FUNCTION_BLOCK C_BINARYREADER
VAR_INPUT
END_VAR
VAR_OUTPUT
END_VAR
VAR
	_BASESTREAM 	: I_STREAM;
END_VAR

PROPERTY BASE_STREAM : I_STREAM
GET
Base_Stream := _BASESTREAM;
END_GET
END_PROPERTY

METHOD CLOSE : DINT
VAR_INPUT
END_VAR
Close := _BASESTREAM.Close();
_BASESTREAM := 0;
RETURN;
END_METHOD

METHOD NEW : DINT
VAR_INPUT
	STREAM : I_STREAM;
END_VAR
IF STREAM = 0 THEN
	New := 1;
	RETURN;
ELSE
	IF STREAM.IsValid THEN
		_BASESTREAM := STREAM;
		_BASESTREAM.Seek( 0, E_STREAMSEEKTYPE.Origin);
		New := -1;
		RETURN;
	ELSE
		New := 1;
		RETURN;
	END_IF
END_IF
END_METHOD

METHOD READ_BOOL : DINT
VAR_INPUT
	out_data : POINTER TO BOOL;
END_VAR
IF _BASESTREAM = 0 THEN
	Read_Bool := 1;
	RETURN;
END_IF

Read_Bool := _BASESTREAM.Read(out_data , 1);
RETURN;
END_METHOD

METHOD READ_BYTES : DINT
VAR_INPUT
	out_data 	: POINTER TO BYTE;
	length		: UDINT;
END_VAR
IF _BASESTREAM = 0 THEN
	Read_Bytes := 1;
	RETURN;
END_IF

Read_Bytes := _BASESTREAM.Read(out_data, length);
RETURN;
END_METHOD

METHOD READ_DOUBLE : DINT
VAR_INPUT
	out_data : POINTER TO LREAL;
END_VAR
IF _BASESTREAM = 0 THEN
	Read_Double := 1;
	RETURN;
END_IF

Read_Double := _BASESTREAM.Read(out_data , 8);
RETURN;
END_METHOD

METHOD READ_FLOAT : DINT
VAR_INPUT
	out_data : POINTER TO REAL;
END_VAR
IF _BASESTREAM = 0 THEN
	Read_Float := 1;
	RETURN;
END_IF

Read_Float := _BASESTREAM.Read(out_data , 4);
RETURN;
END_METHOD

METHOD READ_INT16 : DINT
VAR_INPUT
	out_data : POINTER TO INT;
END_VAR
IF _BASESTREAM = 0 THEN
	Read_Int16 := 1;
	RETURN;
END_IF

Read_Int16 := _BASESTREAM.Read(out_data , 2);
RETURN;
END_METHOD

METHOD READ_INT32 : DINT
VAR_INPUT
	out_data : POINTER TO DINT;
END_VAR
IF _BASESTREAM = 0 THEN
	Read_Int32 := 1;
	RETURN;
END_IF

Read_Int32 := _BASESTREAM.Read(out_data , 4);
RETURN;
END_METHOD

METHOD READ_STRING : DINT
VAR_INPUT
	out_data 	: PVOID;
	length		: UDINT;
END_VAR
IF _BASESTREAM = 0 THEN
	Read_String := 1;
	RETURN;
END_IF

Read_String := _BASESTREAM.Read(out_data, length);
RETURN;
END_METHOD

METHOD READ_UINT16 : DINT
VAR_INPUT
	out_data : POINTER TO UINT;
END_VAR
IF _BASESTREAM = 0 THEN
	Read_UInt16 := 1;
	RETURN;
END_IF

Read_UInt16 := _BASESTREAM.Read(out_data , 4);
RETURN;
END_METHOD

METHOD READ_UINT32 : DINT
VAR_INPUT
	out_data : POINTER TO UDINT;
END_VAR
IF _BASESTREAM = 0 THEN
	Read_UInt32 := 1;
	RETURN;
END_IF

Read_UInt32 := _BASESTREAM.Read(out_data , 4);
RETURN;
END_METHOD

END_FUNCTION_BLOCK

(* stored: Version 1.1.0.1, ProductVersion 3.1.4020.3
   POU C_BINARYREADER: Id {3b66d005-3f47-4af4-a375-894516dc8bea}, SpecialFunc None
   Property BASE_STREAM: Id {71cc1926-e2dc-417b-be5f-3e2a654df2aa}
   Get Get: Id {e0c76d2d-5cef-40c9-82e4-8af46b1fce9d}
   Method CLOSE: Id {de3cb16b-5206-41f8-a6b6-71c7bc0eb741}
   Method NEW: Id {4608d601-859c-47f4-831c-e01655b347f4}
   Method READ_BOOL: Id {76d45542-60ae-421d-a421-b25cd500e521}
   Method READ_BYTES: Id {369d9618-2206-40c5-ad7f-cfb8812abbed}
   Method READ_DOUBLE: Id {db11d57f-7dd3-4a73-85f8-532f0941f54f}
   Method READ_FLOAT: Id {44748d10-e06c-4cd0-983b-1dae6ee03d82}
   Method READ_INT16: Id {2b50ad5d-6d0a-4a08-a27e-1dee1b4acca2}
   Method READ_INT32: Id {555c708b-06af-4983-bc95-ad72bfff7519}
   Method READ_STRING: Id {8bbb68ff-c92f-4a55-8401-1cce0167fdf4}
   Method READ_UINT16: Id {73cf70b9-22f9-426b-a7d1-458ae4cb6acc}
   Method READ_UINT32: Id {b9ecc356-b187-4340-98f9-de3663fa31b7} *)
